{attribute 'linkalways'} 
{attribute 'no_explicit_call' := 'This FB is a CLASS and must be accessed using methods or properties'}
{attribute 'enable_dynamic_creation'}
FUNCTION_BLOCK Node_F_VN_CheckIfEmpty EXTENDS VisionNode
VAR
    ipContainer : _ITcVnContainer;
    hrPrev : _HRESULT(S_OK);
	hresult : _HRESULT(S_OK);
END_VAR

METHOD PUBLIC  Clone : I_Node
VAR
	pNode : POINTER TO Node_F_VN_CheckIfEmpty;
END_VAR
pNode := __NEW(Node_F_VN_CheckIfEmpty);
Clone := pNode^;
END_METHOD

METHOD FB_init : BOOL
VAR_INPUT
	bInitRetains : BOOL; // if TRUE, the retain variables are initialized (warm start / cold start)
	bInCopyCode : BOOL;  // if TRUE, the instance afterwards gets moved into the copy code (online change)
END_VAR
AddInput('ipContainer', ipContainer);
AddInput('hrPrev', hrPrev);
AddOutput('hresult',hresult);
END_METHOD

METHOD PROTECTED OnExecute
hresult.Value := F_VN_CheckIfEmpty(
	ipContainer := ipContainer.Value,
	hrPrev:= hrPrev.Value);
END_METHOD

METHOD PUBLIC PreExecutionCheck
VAR_INPUT
	Check : I_PreExecutionChecks;
END_VAR
Check.IsTrue(ipContainer.IsValid, 'ipContainer must be a valid container');
END_METHOD

END_FUNCTION_BLOCK

(* stored: Version 1.1.0.1, ProductVersion 3.1.4024.13
   POU Node_F_VN_CheckIfEmpty: Id {46badf94-e7d7-0cb0-356f-ef0bb0a09bf5}, SpecialFunc None
   Folder Constructor: Id {927a795f-ce17-0914-0208-466c6d5931ae}
   Method Clone: Id {32d02d97-e61f-0bcc-191a-59bc39291428}
   Method FB_init: Id {962c190e-16d0-0270-3e18-deea4bffa0d4}
   Method OnExecute: Id {8bff8fc1-e066-0d92-2296-8bd422c0ce54}
   Method PreExecutionCheck: Id {436f9fee-4c2e-0c62-0fec-7df00d79929f} *)
